// TIA Portal V16 export
// export: Created 2026-03-31T12:42:57.7280988Z, ExportSetting WithDefaults, DisplayName Totally Integrated Automation Portal, DisplayVersion V16, DisplayName TIA Portal Version Control Interface, DisplayVersion V16, DisplayName TIA Portal Openness, DisplayVersion V16, DisplayName STEP 7 Professional, DisplayVersion V16, DisplayName STEP 7 Safety, DisplayVersion V16, DisplayName WinCC Advanced, DisplayVersion V16
ORGANIZATION_BLOCK "OB121"   // OB121, FBD, ProgrammingError
VERSION : 0.1
// stored: IsIECCheckEnabled false
   VAR_TEMP
      Temp_0 : Byte;
      Temp_1 : Byte;
      Temp_2 : Byte;
      Temp_3 : Byte;
      Temp_4 : Byte;
      Temp_5 : Byte;
      Temp_6 : Word;
      Temp_7 : Word;
      Temp_8 : Word;
      Temp_9 : Date_And_Time;
   END_VAR
BEGIN
END_ORGANIZATION_BLOCK
